# B&R Automation Studio project develop
Automation Studio 4.3.6.57 SP; technology packages: Acp10Arnc0 3.18.2

## Configuration ARM

CPU X20CP0410, AutomationRuntime B4.63, Build 4.1.2, Vc V4.62.0

### Task classes (Cpu.sw)
```
Cyclic#4 (cycle 100000 us, tolerance 100000 us):
  P76C <- P76Sample.P76C.prg
DataObjects: P76config <- Parameter.P76config.dob
Binaries: FWRules, udbdef, TCData, ashwd, ashwac, asfw, iomap, sysconf, Role, User, arconfig
Libraries: Operator, Runtime, AsTime, AsIecCon, brsystem, DataObj, sys_lib, ac_invlib, AsArLog, AsCANopen, AsBrStr, FileIO, AsBrMath, AsEPL
```

### Hardware
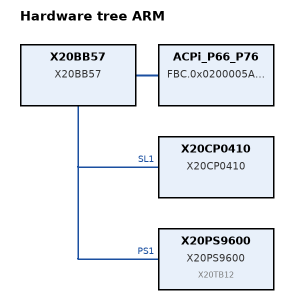
```
ACPi_P66_P76 : FBC.0x0200005A.320.ACPi_P66_P76 v1.3 (OrderNumber=ACPi_P66_P76)  [CAN1 -> X20BB57.IF7]
X20BB57 : X20BB57 v1.1.0.0
  Connector IF7:
    Baudrate = 250000
    ActivateCANIO = 0
    ActivateCanOpen = 1
    p100c_parametervalue = 1000
    p100d_parametervalue = 3
X20CP0410 : X20CP0410 v1.2.0.0  [SL -> X20BB57.SL1]
  Connector IF2:
    ActivateDevice = 1
    Mode = Manual
    InternetAddress = 192.168.0.35
    SubnetMask = 255.255.255.0
  ConfigurationID = develop_ARM
  TimerDeviceType = SWIOTIMER
  Cyclic1Duration = 10000
  Cyclic1Tolerance = 10000
  Cyclic2Duration = 20000
  Cyclic2Tolerance = 20000
  Cyclic3Duration = 50000
  Cyclic3Tolerance = 50000
  Cyclic4Duration = 100000
  Cyclic4Tolerance = 100000
  Cyclic5Duration = 200000
  Cyclic5Tolerance = 200000
  Cyclic6Duration = 500000
  Cyclic6Tolerance = 500000
  Cyclic7Duration = 1000000
  Cyclic7Tolerance = 1000000
  Cyclic8Duration = 10000
  Cyclic8Tolerance = 30000000
X20PS9600 : X20PS9600 v1.2.0.0  [PS -> X20BB57.PS1; SS1 -> X20TB12.SS]
X20TB12 : X20TB12 v1.0.0.0
```

### IoMap.iom - X20CP0410/IoMap.iom
```iecst
VAR_CONFIG
	::P76C:ac_inv_alloc_0.io_mapping.ModuleOK AT %IX."ACPi_P66_P76".ModuleOk;
	::P76C:ac_inv_alloc_0.io_mapping.LCR AT %IW."ACPi_P66_P76".LCR_2002sub5;
	::P76C:ac_inv_alloc_0.io_mapping.OTR AT %IW."ACPi_P66_P76".OTR_2002sub6;
	::P76C:ac_inv_alloc_0.io_mapping.THD AT %IW."ACPi_P66_P76".THD_2002suba;
	::P76C:ac_inv_alloc_0.io_mapping.HMIS AT %IW."ACPi_P66_P76".HMIS_2002sub29;
	::P76C:ac_inv_alloc_0.io_mapping._LFT AT %IW."ACPi_P66_P76".LFT_2029sub16;
	::P76C:ac_inv_alloc_0.io_mapping.THR AT %IW."ACPi_P66_P76".THR_2042sub1f;
	::P76C:ac_inv_alloc_0.io_mapping.CMDD AT %QW."ACPi_P66_P76".CMDD_6040;
	::P76C:ac_inv_alloc_0.io_mapping.ETAD AT %IW."ACPi_P66_P76".ETAD_6041;
	::P76C:ac_inv_alloc_0.io_mapping.LFRD AT %QW."ACPi_P66_P76".LFRD_6042;
	::P76C:ac_inv_alloc_0.io_mapping.RFRD AT %IW."ACPi_P66_P76".RFRD_6044;
END_VAR
```

## Configuration ATOM

CPU X20CP3585, AutomationRuntime L4.10, Build 2.95.3, Vc V4.15.9

### Task classes (Cpu.sw)
```
Cyclic#4:
  P84 <- P84Sample.P84.prg
  P74 <- P74Sample.P74.prg
DataObjects: P84config <- P84Sample.P84config.dob, P74config <- P74Sample.P74config.dob, Acp10sys
Binaries: udbdef, ashwac, ashwd, sysconf, asfw, arconfig, iomap, Acp10cfg, Acp10map, NeueNcMap
Libraries: brsystem, DataObj, sys_lib, ac_invlib, AsEPL, AsArLog, AsBrStr, AsBrMath, Operator, Runtime, AsTime, AsIecCon, asstring, AsCANopen, FileIO, powerlnk, ncglobal, AsUSB, acp10sdc, wh_regl, acp10sim, wh_aclib, acp10par, acp10man
```

### Hardware
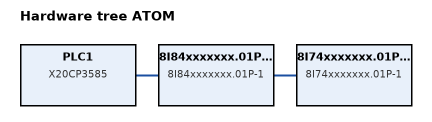
```
8I74xxxxxxx.01P-1 : 8I74xxxxxxx.01P-1 v1.4.0.0  [PLK1 -> 8I84xxxxxxx.01P-1.PLK2 (NodeNumber=10) [Cable Type=PowerlinkCable, Length=10, Version=1.0.0.1]]
  Supervision = off
  packedETAD = packed
  packedETI = packed
  packedCMDD = packed
  packedCMI = packed
  DownloadParameters = no
  ACC = 10
  DEC = 10
8I84xxxxxxx.01P-1 : 8I84xxxxxxx.01P-1 v1.0.9.2  [PLK1 -> PLC1.IF3 (NodeNumber=4) [Cable Type=PowerlinkCable, Length=10, Version=1.0.0.1]; PLK2 -> 8I74xxxxxxx.01P-1.PLK1 (NodeNumber=4) [Cable Type=PowerlinkCable, Length=10, Version=1.0.0.1]]
  Supervision = off
  packedETAD = packed
  packedETI = packed
  packedCMDD = packed
  packedCMI = packed
  DownloadParameters = no
  AUT = 1
PLC1 : X20CP3585 v1.4.2.0
  Connector IF2:
    ActivateDevice = 1
    Mode = Manual
    InternetAddress = 192.168.0.10
    SubnetMask = 255.255.255.0
  Connector IF3:
    InaNodeNumber = 1
  ConfigurationID = develop_ATOM
```

### IoMap.iom - PLC1/IoMap.iom
```iecst
(********************************************************************
 * COPYRIGHT -- Bernecker + Rainer
 ********************************************************************
 * File: IoMap.iom
 * Author: hilchenbachc
 * Created: September 05, 2012
 ********************************************************************
 * IO mapping file
 ********************************************************************)
VAR_CONFIG
	::P84:ac_inv_alloc_0.io_mapping.ModuleOK AT %IX."8I84xxxxxxx.01P-1".ModuleOk;
	P84:ac_inv_alloc_0.io_mapping.ETAD AT %IW."8I84xxxxxxx.01P-1".ETAD_Input;
	P84:ac_inv_alloc_0.io_mapping.HMIS AT %IW."8I84xxxxxxx.01P-1".HMIS_Input;
	P84:ac_inv_alloc_0.io_mapping.LCR AT %IW."8I84xxxxxxx.01P-1".LCR_Input;
	P84:ac_inv_alloc_0.io_mapping.THD AT %IW."8I84xxxxxxx.01P-1".THD_Input;
	P84:ac_inv_alloc_0.io_mapping.THR AT %IW."8I84xxxxxxx.01P-1".THR_Input;
	P84:ac_inv_alloc_0.io_mapping.CMDD AT %QW."8I84xxxxxxx.01P-1".CMDD_Output;
	P84:ac_inv_alloc_0.io_mapping.CMI AT %QW."8I84xxxxxxx.01P-1".CMI_Output;
	P84:ac_inv_alloc_0.io_mapping.LFRD AT %QW."8I84xxxxxxx.01P-1".LFRD_Output;
	P84:ac_inv_alloc_0.io_mapping.LTR AT %QW."8I84xxxxxxx.01P-1".LTR_Output;
	P84:ac_inv_alloc_0.io_mapping.LFT AT %IW."8I84xxxxxxx.01P-1".LFT_Input;
	P84:ac_inv_alloc_0.io_mapping.RFRD AT %IW."8I84xxxxxxx.01P-1".RFRD_Input;
	P84:ac_inv_alloc_0.io_mapping.OTR AT %IW."8I84xxxxxxx.01P-1".OTR_Input;
	P74:ac_inv_alloc_0.io_mapping.ETAD AT %IW."8I74xxxxxxx.01P-1".ETAD_Input;
	P74:ac_inv_alloc_0.io_mapping.HMIS AT %IW."8I74xxxxxxx.01P-1".HMIS_Input;
	P74:ac_inv_alloc_0.io_mapping.LCR AT %IW."8I74xxxxxxx.01P-1".LCR_Input;
	P74:ac_inv_alloc_0.io_mapping.RFRD AT %IW."8I74xxxxxxx.01P-1".RFRD_Input;
	P74:ac_inv_alloc_0.io_mapping.OTR AT %IW."8I74xxxxxxx.01P-1".OTR_Input;
	P74:ac_inv_alloc_0.io_mapping.THD AT %IW."8I74xxxxxxx.01P-1".THD_Input;
	P74:ac_inv_alloc_0.io_mapping.THR AT %IW."8I74xxxxxxx.01P-1".THR_Input;
	P74:ac_inv_alloc_0.io_mapping.LFT AT %IW."8I74xxxxxxx.01P-1".LFT_Input;
	P74:ac_inv_alloc_0.io_mapping.CMDD AT %QW."8I74xxxxxxx.01P-1".CMDD_Output;
	P74:ac_inv_alloc_0.io_mapping.CMI AT %QW."8I74xxxxxxx.01P-1".CMI_Output;
	P74:ac_inv_alloc_0.io_mapping.LFRD AT %QW."8I74xxxxxxx.01P-1".LFRD_Output;
	P74:ac_inv_alloc_0.io_mapping.ModuleOK AT %IX."8I74xxxxxxx.01P-1".ModuleOk;
END_VAR
```

## Logical view

Binary libraries used (declarations not repeated): operator, runtime, AsTime, AsIecCon, brsystem, DataObj, sys_lib, asstring, AsEPL, AsArLog, AsCANopen, AsBrStr, FileIO, AsBrMath

### Package Logical/Libraries - Global libraries

### Library Logical/Libraries/ac_invlib (ANSIC, version 1.10.1) - ACOPOSinverter Library - controls an ACOPOSinverter drive without using the SDC- Library
Depends on: AsEPL, sys_lib, DataObj, AsArLog, brsystem, AsCANopen

#### ac_invlib.typ - Exported data types
```iecst
(********************************************************************
 * COPYRIGHT -- Bernecker + Rainer
 ********************************************************************
 * Library: wh_invlib
 * File: wh_invlib.typ
 * Author: hilchenbachc
 * Created: December 03, 2009
 ********************************************************************
 * Data types of library wh_invlib
 ********************************************************************)

TYPE
	ac_inv_AxIdent : 	STRUCT  (*(internal data type for debugging only !)*)
		p_alloc : REFERENCE TO ac_inv_alloc; (*pointer to fub instance*)
		step_init : UINT; (*initialization step*)
		errorstep : UINT; (*step in which the internal error occured*)
		step_read_data : UINT; (*step for reading data from drive*)
		fub_sdoread : EplSDORead; (*fub instance*)
		fub_sdowrite : EplSDOWrite; (*fub instance*)
		fub_canopen_sdoread : CANopenSDOReadData; (*fub instance*)
		fub_canopen_sdowrite : CANopenSDOWriteData; (*fub instance*)
		node_number : USINT; (*powerlink node number or canopen node number of inverter*)
		interface : STRING[20]; (*interface name*)
		ctrl_on_internal : BOOL; (*internal command for 'ctrl_on'*)
		sdo_read_step : UINT; (*SDORead: step and command interface*)
		sdo_read_par_name : STRING[10]; (*SDORead: name of the inverter parameter*)
		sdo_read_value : UINT; (*SDORead: numeric parameter value*)
		sdo_read_value_constant : STRING[20]; (*SDORead: parameter value constant*)
		sdo_read_status : UINT; (*SDORead: status result*)
		sdo_read_errorinfo : UDINT; (*SDORead: additional error information*)
		sdo_write_step : UINT; (*SDOWrite: step and command interface*)
		sdo_write_par_name : STRING[10]; (*SDOWrite: name of the inverter parameter*)
		sdo_write_value : UINT; (*SDOWrite: numeric parameter value*)
		sdo_write_value_constant : STRING[20]; (*SDOWrite: parameter value constant*)
		sdo_write_status : UINT; (*SDOWrite: status result*)
		sdo_write_errorinfo : UDINT; (*SDOWrite: additional error information*)
		fub_datobjinfo : DatObjInfo; (*fub instance*)
		number_of_parameters : UDINT; (*number of parameters in dataobject*)
		parameterlist_index : UINT; (*parameter list: index of the actual parameter*)
		p_sorted_parameters : ARRAY[0..99]OF UDINT; (*pointer to list with the sorted parameters*)
		dont_sort_parameters : BOOL; (*don't sort parameters from datamodules*)
		write_parameterlist_step : UINT; (*write parameter list: step and command interface*)
		write_parameterlist_status : UINT; (*write parameter list: status result*)
		compare_parameterlist_step : UINT; (* Compare paameterlist: step and command interface *)
		compare_parameterlist_status : UINT; (* Compare parameterlist: status result *)
		compare_parameterlist_index : USINT; (* compare parameterlist: index of the actual parameter *)
		compare_value_constant : STRING[20]; (*SDORead: parameter value constant*)
		log_info : STRING[60]; (*row in logging information*)
		fub_log_write : AsArLogWrite; (*fub instance*)
		kv_old : UINT; (*gain speed controller in %*)
		ti_old : UINT; (*integral time speed controller in %*)
		counter_cyclic_data : USINT; (*cycle counter for cyclic read data*)
		HMIS_old : INT;
		rated_motor_frequency : REAL; (*FrS*)
		rated_motor_speed : REAL; (*nSP*)
		maximum_output_frequency : REAL; (*tFr*)
		polepairs : USINT; (*no of motor polepairs*)
		use_rpm : BOOL; (*1 = use rpm instead Hertz for motor speeds*)
		t_limit_old : ARRAY[0..1]OF REAL;
		cycleTime : REAL; (*cycle time of the task*)
		timer : REAL; (*timer for waiting actions*)
		device_name : STRING[20]; (*Device- Name from Powerlink Object 0x1008*)
		drive_type : USINT; (*0 = unknown, 1 = P84, 2 = P74*)
		isCANopen : BOOL; (*1 = is a CANopen- device*)
		tempUINT : UINT;
	END_STRUCT;
	ac_inv_Mapping : 	STRUCT
		ModuleOK : BOOL; (*Module OK (from drive)*)
		ETAD : UINT; (*Status Word (from drive)*)
		HMIS : UINT; (*Drive state Input (from drive)*)
		RFRD : INT; (*Output- velocity (from drive)*)
		OTR : INT; (*Motor torque (from drive)*)
		LCR : UINT; (*Drive Current (from drive)*)
		THD : UINT; (*Drive Thermal State (from drive)*)
		THR : UINT; (*Motor Thermal State (from drive)*)
		LFT : INT; (*Fault Code ( from drive) as INT for EPL-Mapping*)
		_LFT : UINT; (*Fault Code ( from drive) as UINT for CANopen-Mapping (P84 only)*)
		CMDD : UINT; (*Control Word (to drive)*)
		CMI : UINT; (*Extended Control Word (to drive)*)
		LFRD : INT; (*Speed setpoint (to drive)*)
		LTR : INT; (*Torque setpoint (to drive) (P84 only)*)
	END_STRUCT;
END_TYPE
```

#### ac_invlib.var - Exported constants
```iecst
VAR CONSTANT
	ac_invlibERR_CFI : UINT := 50005; (*one or more parameter were corrected by the drive due to consistency check*)
	ac_invlibERR_WRONG_ARVERSION : UINT := 50003; (*wrong Automation Runtime version*)
	ac_invlibERR_PARNOTFOUND : UINT := 50002; (*wrong parameter name*)
	ac_invlibERR_ILLEGAL_AXIDENT : UINT := 50001; (*invalid ax_ident*)
	ac_invlibERR_NETWORK : UINT := 50004; (*network timeout*)
END_VAR
```

#### ac_invlib.fun - Exported functions and function blocks
```iecst
FUNCTION_BLOCK ac_inv_alloc (*axis allocation*)
	VAR_INPUT
		pDevice : UDINT; (*pointer to name of device i.e. 'IF3.ST4'*) (* *) (*#PAR*)
		pcfgpar : ARRAY[0..2] OF UDINT; (*pointer to name of parameter data objects*) (* *) (*#PAR*)
		io_mapping : ac_inv_Mapping; (*IO- mapping (must be connected in physical view)*) (* *) (*#PAR*)
		rpm : BOOL; (*use rpm instead of Hertz for n_set and n_act*) (* *) (*#PAR#OPT*)
		no_parameter_sort : BOOL; (*1 = don't sort parameters from datamodules*) (* *) (*#PAR#OPT*)
	END_VAR
	VAR_OUTPUT
		status : UINT; (*fub status*) (* *) (*#CYC*)
		message : STRING[80]; (*error message, when allocation fails*) (* *) (*#CYC*)
		ax_ident : UDINT; (*axis identifier ('handle') for function blocks*) (* *) (*#CYC*)
	END_VAR
END_FUNCTION_BLOCK

FUNCTION_BLOCK ac_inv (*cyclic execution*)
	VAR_INPUT
		ax_ident : UDINT; (*axis identifier (handle) from ac_inv_alloc()*) (* *) (*#PAR*)
		quickstop : BOOL; (*0 = perform fast stop*) (* *) (*#CMD*)
		ctrl_on : BOOL; (*switch controller (power stage) on/off*) (* *) (*#CMD*)
		f_quit : BOOL; (*quit inverter fault*) (* *) (*#CMD*)
		kv : UINT; (*gain speed controller in %*) (* *) (*#OPT#CYC*)
		ti : UINT; (*Integral time speed controller in %*) (* *) (*#OPT#CYC*)
		n_set : REAL; (*set speed (% of tFr or rpm)*) (* *) (*#CYC*)
		t_set : REAL; (*set torque in % nominal motor torque (P84 only)*) (* *) (*#OPT#CYC*)
		t_limit : ARRAY[0..1] OF REAL; (*torque limit*) (* *) (*#OPT#CYC*)
		write_parameter : USINT; (*write a parameter to the drive (see 'parameter_name' and 'parameter_value')*) (* *) (*#CMD#OPT*)
		read_parameter : USINT; (*read a parameter from the drive (see 'parameter_name' and 'parameter_value')*) (* *) (*#CMD#OPT*)
		parameter_name : STRING[4]; (*name of the inverter parameter to be written or to be read*) (* *) (*#PAR#OPT*)
		parameter_value : STRING[15]; (*value of the inverter parameter to be written or to be read*) (* *) (*#CMD#OPT*)
		C211 : BOOL; (*Control Bit*) (* *) (*#OPT#CYC*)
		C212 : BOOL; (*Control Bit*) (* *) (*#OPT#CYC*)
		C213 : BOOL; (*Control Bit*) (* *) (*#OPT#CYC*)
		C214 : BOOL; (*Control Bit*) (* *) (*#OPT#CYC*)
		C215 : BOOL; (*Control Bit*) (* *) (*#OPT#CYC*)
		activate_tuning : BOOL; (*1 = set motor tuning active. tuning will be activated with 'ctrl_on=true'*) (* *) (*#OPT#CYC*)
	END_VAR
	VAR_OUTPUT
		ctrl_ready : BOOL; (*controller is ready to be switched on*) (* *) (*#CYC*)
		power_line : BOOL; (*power line present = 1*) (* *) (*#CYC*)
		ctrl_is_on : BOOL; (*controller (power stage) is on/off*) (* *) (*#CYC*)
		initialized : BOOL; (*drive initialized*) (* *) (*#CYC*)
		alarm : BOOL; (*alarm*) (* *) (*#CYC*)
		fault : BOOL; (*inverter fault see 'fault code'*) (* *) (*#CYC*)
		PRA_detected : BOOL; (*Power removal (PRA) was detected -> reset ctrl_on*) (* *) (*#CYC#OPT*)
		n_act : REAL; (*actual speed (% of tFr or rpm)*) (* *) (*#CYC*)
		t_act : REAL; (*torque in % of nominal motor torque*) (* *) (*#CYC*)
		current : REAL; (*current in A*) (* *) (*#CYC*)
		thst_drive : REAL; (*thermal state drive in %*) (* *) (*#CYC#OPT*)
		thst_motor : REAL; (*thermal state motor in %*) (* *) (*#CYC*)
		udc : REAL; (*dc voltage in V*) (* *) (*#CYC*)
		encoder_value : UINT; (*encoder value (P84 only)*) (* *) (*#CYC#OPT*)
		drive_state : STRING[4]; (*drive state*) (* *) (*#CYC*)
		fault_code : STRING[4]; (*fault code (LFT) as string*) (* *) (*#CYC*)
		LFT : UINT; (*LFT*) (* *) (*#CYC*)
		status : UINT; (*fub status*) (* *) (*#CYC*)
	END_VAR
END_FUNCTION_BLOCK
```

#### ac_inv_global.h
```c
#ifndef _AC_INV_GLOBAL_H
#define _AC_INV_GLOBAL_H

#include <bur/plctypes.h>
#include <ac_invlib.h>
#include <ctype.h>
#include <string.h>
#include <math.h>

#define STEP_W_NETWORK					0
#define STEP_READ_DEVICE_NAME			1
#define STEP_LOG_DEVICE_TYPE			200
#define STEP_W_LOG_DEVICE_TYPE			201
#define STEP_W_FACTORY_RESET_P74		202
#define STEP_W_P74_CONFIG_1				203
#define STEP_W_P74_CONFIG_2				204
#define STEP_W_FACTORY_RESET_P84		3
#define STEP_W_P84_CONFIG_1				4
#define STEP_W_P84_CONFIG_2				5
#define STEP_W_REFERENCE_CHANNEL_SET 	9
#define STEP_W_PARAMETER_LIST_DOWNLOAD	10
#define STEP_CHECK_PARAMETER_LIST		20
#define STEP_W_PARAMETER_LIST_CHECKED	22
#define STEP_READ_KV					30
#define STEP_READ_TI					31
#define STEP_READ_OUTPUT_FREQUENCY		32
#define STEP_READ_TORQUE_LIMIT_0		33
#define STEP_READ_TORQUE_LIMIT_1		34
#define STEP_READ_CTT					40
#define STEP_READ_RATED_FREQ			41
#define STEP_READ_RATED_SPEED			42
#define STEP_W_READ_RATED_SPEED			43
#define STEP_W_COMMAND					100
#define STEP_P84_WRITE_TUN				300
#define STEP_W_P84_TUNING_DONE			310
#define STEP_P74_START_TUNING			350
#define STEP_P74_TUNING_1				360
#define STEP_P74_TUNING_2				361
#define STEP_P74_TUNING_3				362
#define STEP_P74_TUNING_4				363
#define STEP_P74_TUNING_5				364
#define STEP_P74_TUNING_6				365
#define STEP_P74_TUNING_7				366
#define STEP_P74_TUNING_8				367

#define STEP_INTERNAL_ERROR				9999

char * m_ltoa(long value, char *string, int radix);
long m_atol(char*);
/*int strcasecmp( char *s1, char *s2 );*/
int find_parameter( char *name, UINT *index, USINT *subindex, USINT drive_type );
int find_download_index( char *name,  USINT drive_type );
char *find_value_constant( char *name, UINT value, USINT drive_type );
int find_numeric_value( char *name, char *constant, USINT drive_type );
void read_parameter( ac_inv_AxIdent *ax_ident );
void write_parameter( ac_inv_AxIdent *ax_ident );
void write_parameterlist( ac_inv_AxIdent *ax_ident );
void compare_parameterlist( ac_inv_AxIdent *ax_ident );
void logCOF( ac_inv_AxIdent *ax_ident );
void sort_parameterlist( ac_inv_AxIdent *ax_ident );
void create_parameterlist( ac_inv_AxIdent *ax_ident );
#endif
```

#### ac_invhelp.c
```c
#include <bur/plctypes.h>
#include <ctype.h>

/* long to ascii conversion */
char * m_ltoa(long value, char *string, int radix)
{
  char tmp[33];
  char *tp = tmp;
  long i;
  unsigned long v;
  int sign;

  if (radix > 36 || radix <= 1)
  {
    return 0;
  }

  sign = (radix == 10 && value < 0);
  if (sign)
    v = -value;
  else
    v = (unsigned long)value;
  while (v || tp == tmp)
  {
    i = v % radix;
    v = v / radix;
    if (i < 10)
      *tp++ = i+'0';
    else
      *tp++ = i + 'a' - 10;
  }

  if (sign)
    *string++ = '-';
  while (tp > tmp)
    *string++ = *--tp;
  *string = 0;
  return string;
}

long m_atol( char* s ){
	long l = 0;
	int sign = 0;

	while( *s ){
		if( *s  == '-' ){
			if( sign == 0 )
				sign = -1;
			else
				return 0; /* error: more than one sign */
		}
		if( *s == '+' ){
			if( sign == 0 )
				sign = +1;
			else
				return 0; /* error: more than one sign */
		}
		if( *s >= '0' && *s <= '9' ){
			l *= 10;
			l += *s - '0';
		}
		++s;
	}
	if( sign < 0 )
		l = -l;
	return l;
}

/* case insensitive string comparator */
int strcasecmp( char *s1, char *s2 ){
	do{
		if( tolower( *s1 ) != tolower( *s2 ) ){
			return ( *s1 - *s2 );
		}
		++s1;
		++s2;
	} while (*s1 && *s2);
	if( *s1 != *s2 ) /* different length */
		return -1;

	return 0;
}
```

#### ac_invparameter.c
```c
#include <bur/plctypes.h>
#include <stdlib.h>
#include <string.h>
#include <ac_inv_global.h>

#include <ac_invparameter.h>
#include <P84_registers.h>
#include <P74_registers.h>

/* -----------------------------------------------------------------------------------
   find parameter in list
   returns index of parameter in parameter list or -1 in case of failure
   -----------------------------------------------------------------------------------
*/

int find_parameter( char *name, UINT *index, USINT *subindex, USINT drive_type )
{
	int i = 0;
	acpireg *regs = drive_type == 2 ? p74reg : p84reg;

	while( regs[i].name )
	{
		if( strcasecmp( regs[i].name, name ) == 0 )   /* found ? */
		{
			if( index )
				*index = regs[i].index;
			if( subindex )
				*subindex = regs[i].subindex;
			return i;
		}
		++i;
	}
	return -1; /* not found */
}

/* -----------------------------------------------------------------------------------
 	returns the download index of a parameter or -1 in case of failure
   -----------------------------------------------------------------------------------
*/

int find_download_index( char *name,  USINT drive_type )
{
	int i = 0;
	char **list = drive_type == 2 ? P74_download_index : P84_download_index;

	while( list[i] )
	{
		if( strcasecmp(  list[i], name ) == 0 )   /* found ? */
		{
			return i;
		}
		++i;
	}
	return -1; /* not found */
}

/* -----------------------------------------------------------------------------------
 	returns the enumerated name of the parameter's value
   -----------------------------------------------------------------------------------
*/

char *find_value_constant( char *name, UINT value, USINT drive_type )
{
	int index;
	static char s[20];
	char sign = 'u';
	acpireg *regs = drive_type == 2 ? p74reg : p84reg;

	index = find_parameter( name, 0, 0, drive_type );
	if( index >= 0 )
	{
		int i = 0;
		sign = regs[index].sign;
		/* translate parameter value to enumeration constant */
		if( regs[index].enu )   /* are constants defined ? */
		{
			while( regs[index].enu[i].name )
			{
				if( regs[index].enu[i].value == value )
				{
					return( regs[index].enu[i].name );  /* return enumerated name */
				}
				++i;
			}
		}
	}
	if( sign == 'u' )
		m_ltoa( value , s, 10 );  /* return numeric value */
	else
		m_ltoa( (INT) value, s, 10 );
	return s; /* not found or no constant defined */

}

/* -----------------------------------------------------------------------------------
 	returns the value for the given constant
   -----------------------------------------------------------------------------------
*/

int find_numeric_value( char *name, char *constant, USINT drive_type )
{
	int index;
	acpireg *regs = drive_type == 2 ? p74reg : p84reg;

	index = find_parameter( name, 0, 0, drive_type );
	if( index >= 0 )
	{
		int i = 0;
		/* try to find the constant */
		if( regs[index].enu )   /* are constants defined ? */
		{
			while( regs[index].enu[i].name )
			{
				if( strcasecmp( regs[index].enu[i].name, constant ) == 0 )
				{
					return( regs[index].enu[i].value );  /* return enumerated name */
				}
				++i;
			}
		}
	}
	return m_atol(constant);  /* return numeric value */

}

/* -------------------------------------------------------------------------------------
   read parameter from inverter
   -------------------------------------------------------------------------------------
*/

void read_parameter( ac_inv_AxIdent *ax_ident )
{

	for(;;)
	{
		switch( ax_ident->sdo_read_step )
		{
		case 0: /* wait for command */
			ax_ident->fub_sdoread.enable = 0;
			break;

		case 1: /* start read */
			if( find_parameter( ax_ident->sdo_read_par_name, &ax_ident->fub_sdoread.index, &ax_ident->fub_sdoread.subindex, ax_ident->drive_type ) < 0 )
			{
				ax_ident->sdo_read_step = 3;
				ax_ident->sdo_read_status = ac_invlibERR_PARNOTFOUND;
				ax_ident->sdo_read_errorinfo = 0;
				continue; /* save on cycle */
			}
			else
			{
				/* fill the fub structure */
				ax_ident->sdo_read_value = 0;
				ax_ident->fub_sdoread.enable = 1;
				ax_ident->fub_sdoread.pData = (UDINT) &ax_ident->sdo_read_value;
				ax_ident->fub_sdoread.datalen = sizeof(ax_ident->sdo_read_value);
				ax_ident->sdo_read_step = 2;
				ax_ident->sdo_read_status = 65535;
				ax_ident->sdo_read_errorinfo = 0;

			}
			break;

		case 2: /* wait until read */
			if( ax_ident->fub_sdoread.status != 65535 )  /* value read */
			{
				ax_ident->fub_sdoread.enable = 0; /* disable fub */
				ax_ident->sdo_read_status = ax_ident->fub_sdoread.status;
				ax_ident->sdo_read_errorinfo = ax_ident->fub_sdoread.errorinfo;
				ax_ident->sdo_read_step = 3;
				continue; /* save on cycle */
			}
			break;

		case 3: /* write into log */
		{
			char tempstring[20];
			const char *ret = find_value_constant( ax_ident->sdo_read_par_name, ax_ident->sdo_read_value, ax_ident->drive_type );
			strcpy( ax_ident->sdo_read_value_constant, ret );
			strcpy( ax_ident->log_info, ax_ident->interface );
			strcat( ax_ident->log_info, "." );
			m_ltoa( ax_ident->node_number, tempstring, 10 );
			strcat( ax_ident->log_info, tempstring );
			strcat( ax_ident->log_info, "  " );
			strcat( ax_ident->log_info, ax_ident->sdo_read_par_name );
			strcat( ax_ident->log_info, " -->#" );
			strcat( ax_ident->log_info, ax_ident->sdo_read_value_constant );
			if( ax_ident->sdo_read_status != 0 )
			{
				ax_ident->fub_log_write.logLevel = arlogLEVEL_FATAL;
				if( ax_ident->sdo_read_status == ERR_ASEPL_ACCESS_FAILED )
				{
					strcat( ax_ident->log_info, ":errorinfo=" );
					strcat( ax_ident->log_info, "/0x" );
					m_ltoa( ax_ident->sdo_read_errorinfo, tempstring, 16 );
					strcat( ax_ident->log_info, tempstring );
				}
				else if( ax_ident->sdo_read_status == ac_invlibERR_PARNOTFOUND )
				{
					strcat( ax_ident->log_info, ":parameter not found" );
				}
			}
			else
			{
				ax_ident->fub_log_write.logLevel = arlogLEVEL_INFO;
			}
			ax_ident->fub_log_write.errornr = ax_ident->sdo_read_status;
			ax_ident->fub_log_write.mem = (UDINT) &ax_ident->node_number;
			ax_ident->fub_log_write.len = sizeof(ax_ident->node_number);
			ax_ident->fub_log_write.asciiString = (UDINT) ax_ident->log_info;
			AsArLogWrite( &ax_ident->fub_log_write );
			ax_ident->sdo_read_step = 4;
		}
		break;

		case 4:  /* wait until log entry written */
			if( ax_ident->fub_log_write.status != 65535 )
			{
				ax_ident->sdo_read_step = 0;
			}
			else
			{
				AsArLogWrite( &ax_ident->fub_log_write );
			}
			break;

			/* start reading without writing to log file in case of success (for fub inside use ! */
		case 10:
			if( find_parameter( ax_ident->sdo_read_par_name, &ax_ident->fub_sdoread.index, &ax_ident->fub_sdoread.subindex, ax_ident->drive_type ) < 0 )
			{
				ax_ident->sdo_read_step = 3;
				ax_ident->sdo_read_status = ac_invlibERR_PARNOTFOUND;
				ax_ident->sdo_read_errorinfo = 0;
				continue; /* save on cycle */
			}
			else
			{
				/* fill the fub structure */
				ax_ident->sdo_read_value = 0;
				ax_ident->fub_sdoread.enable = 1;
				ax_ident->fub_sdoread.pData = (UDINT) &ax_ident->sdo_read_value;
				ax_ident->fub_sdoread.datalen = sizeof(ax_ident->sdo_read_value);
				ax_ident->sdo_read_step = 11;
				ax_ident->sdo_read_status = 65535;
				ax_ident->sdo_read_errorinfo = 0;
			}
			break;

		case 11: /* wait until read */
			if( ax_ident->fub_sdoread.status != 65535 )  /* value read */
			{
				ax_ident->fub_sdoread.enable = 0; /* disable fub */
				ax_ident->sdo_read_status = ax_ident->fub_sdoread.status;
				ax_ident->sdo_read_errorinfo = ax_ident->fub_sdoread.errorinfo;
				ax_ident->sdo_read_step = 0;
			}
			break;

			/* use SDO read directly (for fub inside use !) */
		case 100:
			ax_ident->fub_sdoread.enable = 1;
			ax_ident->sdo_read_step = 101;
			break;

		case 101:
			if( ax_ident->fub_sdoread.status != 65535 )  /* value read */
			{
				ax_ident->fub_sdoread.enable = 0; /* disable fub */
				ax_ident->sdo_read_status = ax_ident->fub_sdoread.status;
				ax_ident->sdo_read_errorinfo = ax_ident->fub_sdoread.errorinfo;
				ax_ident->sdo_read_step = 0;
			}
			break;

		}
		break;  /* exit for(;;) */
	}

	if( ax_ident->isCANopen )
	{
		/* FUB- Eingaenge umkopieren */
		ax_ident->fub_canopen_sdoread.enable = ax_ident->fub_sdoread.enable;
		ax_ident->fub_canopen_sdoread.index = ax_ident->fub_sdoread.index;
		ax_ident->fub_canopen_sdoread.subindex = ax_ident->fub_sdoread.subindex;
		CANopenSDOReadData( &ax_ident->fub_canopen_sdoread );
		/* FUB- Ausgaenge umkopieren */
		ax_ident->fub_sdoread.status = ax_ident->fub_canopen_sdoread.status;
		ax_ident->fub_sdoread.errorinfo = ax_ident->fub_canopen_sdoread.errorinfo;
	}
	else
		EplSDORead( &ax_ident->fub_sdoread );

}

/* -------------------------------------------------------------------------------------
   write parameter to inverter via EPL
   -------------------------------------------------------------------------------------
*/

void write_parameter( ac_inv_AxIdent *ax_ident )
{

	for(;;)
	{
		switch( ax_ident->sdo_write_step )
		{
		case 0: /* wait for command */
			ax_ident->fub_sdowrite.enable = 0;
			break;

		case 1: /* start write */
			if( find_parameter( ax_ident->sdo_write_par_name, &ax_ident->fub_sdowrite.index, &ax_ident->fub_sdowrite.subindex, ax_ident->drive_type ) < 0 )
			{
				ax_ident->sdo_write_step = 3;
				ax_ident->sdo_write_status = ac_invlibERR_PARNOTFOUND;
				ax_ident->sdo_write_errorinfo = 0;
				continue; /* save on cycle */
			}
			else
			{
				/* fill the fub structure */
				ax_ident->sdo_write_value = find_numeric_value( ax_ident->sdo_write_par_name, ax_ident->sdo_write_value_constant, ax_ident->drive_type );
				ax_ident->fub_sdowrite.enable = 1;
				ax_ident->sdo_write_step = 2;
				ax_ident->sdo_write_status = 65535;
				ax_ident->sdo_write_errorinfo = 0;
			}
			break;

		case 2: /* wait until written */
			if( ax_ident->fub_sdowrite.status != 65535 )
			{
				ax_ident->sdo_write_status = ax_ident->fub_sdowrite.status;
				ax_ident->sdo_write_errorinfo = ax_ident->fub_sdowrite.errorinfo;
				ax_ident->fub_sdowrite.enable = 0; /* disable fub */
				ax_ident->sdo_write_step = 3;
				continue; /* save on cycle */
			}
			break;

		case 3: /* write into log */
		{
			char tempstring[20];

			strcpy( ax_ident->log_info, ax_ident->interface );
			strcat( ax_ident->log_info, "." );
			m_ltoa( ax_ident->node_number, tempstring, 10 );
			strcat( ax_ident->log_info, tempstring );
			strcat( ax_ident->log_info, " #" );
			strcat( ax_ident->log_info, ax_ident->sdo_write_value_constant );
			strcat( ax_ident->log_info, " -->" );
			strcat( ax_ident->log_info, ax_ident->sdo_write_par_name );
			if( ax_ident->sdo_write_status != 0 )
			{
				if( ax_ident->sdo_write_status == ERR_ASEPL_ACCESS_FAILED )
				{
					ax_ident->fub_log_write.logLevel = arlogLEVEL_FATAL;
					strcat( ax_ident->log_info, " :errorinfo=" );
					strcat( ax_ident->log_info, "/0x" );
					m_ltoa( ax_ident->sdo_write_errorinfo, tempstring, 16 );
					strcat( ax_ident->log_info, tempstring );
				}
				else if( ax_ident->sdo_write_status == ac_invlibERR_PARNOTFOUND )
				{
					strcat( ax_ident->log_info, ":parameter not found" );
				}
			}
			else
			{
				ax_ident->fub_log_write.logLevel = arlogLEVEL_INFO;
			}
			ax_ident->fub_log_write.errornr = ax_ident->sdo_write_status;
			ax_ident->fub_log_write.mem = (UDINT) &ax_ident->node_number;
			ax_ident->fub_log_write.len = sizeof(ax_ident->node_number);
			ax_ident->fub_log_write.asciiString = (UDINT) ax_ident->log_info;
			AsArLogWrite( &ax_ident->fub_log_write );
			ax_ident->sdo_write_step = 4;
			continue; /* save on cycle */
		}
		break;

		case 4:  /* wait until log entry written */
			if( ax_ident->fub_log_write.status != 65535 )
			{
				ax_ident->sdo_write_step = 0;
			}
			else
			{
				AsArLogWrite( &ax_ident->fub_log_write );
			}
			break;

		}
		break; /* exit for(;;) */
	}

	if( ax_ident->isCANopen )
	{
		/* FUB- Eingaenge umkopieren */
		ax_ident->fub_canopen_sdowrite.enable = ax_ident->fub_sdowrite.enable;
		ax_ident->fub_canopen_sdowrite.index = ax_ident->fub_sdowrite.index;
		ax_ident->fub_canopen_sdowrite.subindex = ax_ident->fub_sdowrite.subindex;
		CANopenSDOWriteData( &ax_ident->fub_canopen_sdowrite );
		/* FUB- Ausgaenge umkopieren */
		ax_ident->fub_sdowrite.status = ax_ident->fub_canopen_sdowrite.status;
		ax_ident->fub_sdowrite.errorinfo = ax_ident->fub_canopen_sdowrite.errorinfo;
	}
	else
		EplSDOWrite( &ax_ident->fub_sdowrite );

}

/* -------------------------------------------------------------------------------------
   write parameter from parameter list to inverter
   -------------------------------------------------------------------------------------
*/

void write_parameterlist( ac_inv_AxIdent *ax_ident )
{
	char tempstring[80];
	char *source, *dest;
	int i;

	switch( ax_ident->write_parameterlist_step )
	{
	case 0:
		break;

	case 1: /* download started - write header to log */
		if( ax_ident->p_alloc->pcfgpar[0] || ax_ident->p_alloc->pcfgpar[1] || ax_ident->p_alloc->pcfgpar[2] )
		{
			ax_ident->parameterlist_index = 0;
			ax_ident->sdo_write_status = 0; /* clear last SDO write error */
			strcpy( ax_ident->log_info, ax_ident->interface );
			strcat( ax_ident->log_info, "." );
			m_ltoa( ax_ident->node_number, tempstring, 10 );
			strcat( ax_ident->log_info, tempstring );
			strcat( ax_ident->log_info, " download " );
			for( i = 0; i < 3; ++i )
			{
				if( ax_ident->p_alloc->pcfgpar[i] )
				{
					strcat( ax_ident->log_info, " \"" );
					strcat( ax_ident->log_info, (char*)	ax_ident->p_alloc->pcfgpar[i] );
					strcat( ax_ident->log_info, "\" " );
				}
			}
			ax_ident->fub_log_write.logLevel = arlogLEVEL_INFO;
			ax_ident->fub_log_write.errornr = 0;
			ax_ident->fub_log_write.mem = (UDINT) &ax_ident->node_number;
			ax_ident->fub_log_write.len = sizeof(ax_ident->node_number);
			ax_ident->fub_log_write.asciiString = (UDINT) ax_ident->log_info;
			AsArLogWrite( &ax_ident->fub_log_write );
			ax_ident->write_parameterlist_step	= 2;
		}
		else
		{
			ax_ident->write_parameterlist_step	= 0;
		}
		break;

	case 2:  /* wait until log entry written */
		if( ax_ident->fub_log_write.status == 0 )
		{
			ax_ident->write_parameterlist_step = 3;
		}
		else if( ax_ident->fub_log_write.status != 65535 )  /* error */
		{
			ax_ident->write_parameterlist_step = 0;
		}
		else
		{
			AsArLogWrite( &ax_ident->fub_log_write );
		}
		break;

	case 3: /* read next row */
		if( ax_ident->sdo_write_step == 0 )   /* service channel free ? */
		{
			source = (char*) ax_ident->p_sorted_parameters[ax_ident->parameterlist_index];
			dest = tempstring;
			memset( tempstring, 0, sizeof(tempstring) );
			if( ax_ident->sdo_write_status != 0 )  /* error after writing the last parameter */
			{
				ax_ident->write_parameterlist_status = ax_ident->sdo_write_status;
				ax_ident->write_parameterlist_step = 0;
				break;
			}
			else if( ax_ident->parameterlist_index >= ax_ident->number_of_parameters )  /* end of list */
			{
				strcpy( ax_ident->log_info, ax_ident->interface );
				strcat( ax_ident->log_info, "." );
				m_ltoa( ax_ident->node_number, tempstring, 10 );
				strcat( ax_ident->log_info, tempstring );
				strcat( ax_ident->log_info, " end of " );
				for( i = 0; i < 3; ++i )
				{
					if( ax_ident->p_alloc->pcfgpar[i] )
					{
						strcat( ax_ident->log_info, " \"" );
						strcat( ax_ident->log_info, (char*)	ax_ident->p_alloc->pcfgpar[i] );
						strcat( ax_ident->log_info, "\" " );
					}
				}
				ax_ident->fub_log_write.logLevel = arlogLEVEL_INFO;
				ax_ident->fub_log_write.errornr = 0;
				ax_ident->fub_log_write.mem = (UDINT) &ax_ident->node_number;
				ax_ident->fub_log_write.len = sizeof(ax_ident->node_number);
				ax_ident->fub_log_write.asciiString = (UDINT) ax_ident->log_info;
				AsArLogWrite( &ax_ident->fub_log_write );
				ax_ident->write_parameterlist_step	= 4;
				break;
			}
			else
			{
				while( ax_ident->parameterlist_index < ax_ident->number_of_parameters )
				{
					if( *source == 0 )   /* end of a row ? */
					{
						strncpy( ax_ident->sdo_write_value_constant, tempstring, sizeof(ax_ident->sdo_write_value_constant) - 1 );
						ax_ident->sdo_write_step = 1;  /* write parameter to inverter */
						++ax_ident->parameterlist_index;
						break;
					}
					else if( !isprint(*source) || *source == ' ' )   /* ignore control chars and spaces */
					{
						++source;
					}
					else if( *source == '=' )
					{
						++source;
						strncpy( ax_ident->sdo_write_par_name, tempstring, sizeof(ax_ident->sdo_write_par_name) - 1 );
						memset( tempstring, 0, sizeof(tempstring) );
						dest = tempstring;
					}
					else
					{
						*dest++ = *source++; /* copy to tempstring */
					}
				}
			}
		}
		break;

	case 4: /* wait until tail is written */
		if( ax_ident->fub_log_write.status != 65535 )
		{
			ax_ident->write_parameterlist_step = 0;
		}
		else
		{
			AsArLogWrite( &ax_ident->fub_log_write );
		}
		break;

	}

}

/* -------------------------------------------------------------------------------------
   compare parameter from parameter list with inverter
   -------------------------------------------------------------------------------------
*/

void compare_parameterlist( ac_inv_AxIdent *ax_ident )
{
	char tempstring[80];
	char *source, *dest;

	switch( ax_ident->compare_parameterlist_step )
	{
	case 0:

		break;

	case 1: /* start comparing */
		ax_ident->parameterlist_index = 0;
		ax_ident->compare_parameterlist_step = 2;
		break;

		/* compare next parameter */
	case 2:
		if( ax_ident->parameterlist_index >= ax_ident->number_of_parameters )  /* end of list */
		{
			ax_ident->compare_parameterlist_step	= 0;
			break;
		}
		else
		{
			source = (char*) ax_ident->p_sorted_parameters[ax_ident->parameterlist_index];
			dest = tempstring;
			memset( tempstring, 0, sizeof(tempstring) );
			while( ax_ident->parameterlist_index < ax_ident->number_of_parameters )
			{
				if( *source == 0 )   /* end of a row ? */
				{
					*dest++ = *source++;
					strncpy( ax_ident->compare_value_constant, tempstring, sizeof(ax_ident->compare_value_constant) - 1 );
					ax_ident->sdo_read_step = 10; /* read without logger entry */
					++ax_ident->parameterlist_index;
					ax_ident->compare_parameterlist_step = 3;
					break;
				}
				else if( !isprint(*source) || *source == ' ' )   /* ignore control chars and spaces */
				{
					++source;
				}
				else if( *source == '=' )
				{
					++source;
					strncpy( ax_ident->sdo_read_par_name, tempstring, sizeof(ax_ident->sdo_read_par_name) - 1 );
					memset( tempstring, 0, sizeof(tempstring) );
					dest = tempstring;
				}
				else
				{
					*dest++ = *source++; /* copy to tempstring */
				}

			}
		}
		break;

		case 3: /* wait for sdo read value */
			if( ax_ident->sdo_read_step == 0 )   /* service channel free ? */
			{
				const char *ret = find_value_constant( ax_ident->sdo_read_par_name, ax_ident->sdo_read_value, ax_ident->drive_type );
				strcpy( ax_ident->sdo_read_value_constant, ret );
				if( strcasecmp( ax_ident->sdo_read_value_constant, ax_ident->compare_value_constant) )  /* different to set value ? */
				{
					ax_ident->compare_parameterlist_step = 4;
				}
				else   /* equal -> ok */
				{
					ax_ident->compare_parameterlist_step = 2;
				}
			}
			break;

		case 4:  /* write into log */
		{
			char tempstring[20];

			strcpy( ax_ident->log_info, ax_ident->interface );
			strcat( ax_ident->log_info, "." );
			m_ltoa( ax_ident->node_number, tempstring, 10 );
			strcat( ax_ident->log_info, tempstring );
			strcat( ax_ident->log_info, "  " );
			strcat( ax_ident->log_info, ax_ident->sdo_read_par_name );
			strcat( ax_ident->log_info, " -->#" );
			strcat( ax_ident->log_info, ax_ident->sdo_read_value_constant );
			strcat( ax_ident->log_info, " (#" );
			strcat( ax_ident->log_info, ax_ident->compare_value_constant );
			strcat( ax_ident->log_info, ")" );
			ax_ident->fub_log_write.logLevel = arlogLEVEL_WARNING;
			ax_ident->fub_log_write.errornr = ac_invlibERR_CFI;
			ax_ident->fub_log_write.mem = (UDINT) &ax_ident->node_number;
			ax_ident->fub_log_write.len = sizeof(ax_ident->node_number);
			ax_ident->fub_log_write.asciiString = (UDINT) ax_ident->log_info;
			AsArLogWrite( &ax_ident->fub_log_write );
			ax_ident->compare_parameterlist_step = 5;
			break;

			case 5:  /* wait until log entry written */
				if( ax_ident->fub_log_write.status != 65535 )
				{
					ax_ident->compare_parameterlist_step = 0;
				}
				else
				{
					AsArLogWrite( &ax_ident->fub_log_write );
				}
			}
			break;

		}

	}

/* -------------------------------------------------------------------------------------
   create a list of parameters from the data modules
   -------------------------------------------------------------------------------------
*/

void create_parameterlist( ac_inv_AxIdent *ax_ident )
{
	int index_module = 0;
	ax_ident->number_of_parameters = 0;
	memset( &ax_ident->p_sorted_parameters, 0, sizeof(ax_ident->p_sorted_parameters) );
	while( ax_ident->p_alloc->pcfgpar[index_module] )
	{
		ax_ident->fub_datobjinfo.enable = 1;
		ax_ident->fub_datobjinfo.pName = ax_ident->p_alloc->pcfgpar[index_module];
		DatObjInfo( &ax_ident->fub_datobjinfo );
		if( ax_ident->fub_datobjinfo.status == 0 )
		{
			char *source = (char*) ax_ident->fub_datobjinfo.pDatObjMem;
			while( ax_ident->fub_datobjinfo.len ){
				if( *source == 0 ){  /* end of a row ? */
					++ax_ident->number_of_parameters;
					while( *source == 0 && ax_ident->fub_datobjinfo.len ){  /* ignore filling zeros */
						++source;
						--ax_ident->fub_datobjinfo.len;
					}
				}
				else if( ax_ident->p_sorted_parameters[ax_ident->number_of_parameters] == 0 ) {  /* store pointer to parameter row */
					ax_ident->p_sorted_parameters[ax_ident->number_of_parameters] = (UDINT) source++;
					ax_ident->fub_datobjinfo.len--;
				}
				else {
					source++;
					ax_ident->fub_datobjinfo.len--;
				}
			}
		}
		if( ++index_module >= 3	)  /* no more data modules */
			break;
	}
}

/* -------------------------------------------------------------------------------------
   compare function for qsort()
   -------------------------------------------------------------------------------------
*/

int compare_download_index_P84 (const void * a, const void * b)
{
	char name[20];
	char *s, *d;
	int index_a=0, index_b=0;
	char **list;

	/* copy parameter name a */
	s = *(char**) a; d= name;
	while( *s != ' ' && *s != 0 && *s != '=')
		*d++ = *s++;
	*d = 0;

	list = P84_download_index;
	while( list[index_a] )
	{
		if( strcasecmp(  list[index_a], name ) == 0 )   /* found ? */
			break;
		++index_a;
	}

	/* copy parameter name b */
	s = *(char**) b; d= name;
	while( *s != ' ' && *s != 0 && *s != '=')
		*d++ = *s++;
	*d = 0;

	list = P84_download_index;
	while( list[index_b] )
	{
		if( strcasecmp(  list[index_b], name ) == 0 )   /* found ? */
			break;
		++index_b;
	}

	if ( index_a <  index_b ) return -1;
	if ( index_a >  index_b ) return 1;

	return 0;
}

int compare_download_index_P74 (const void * a, const void * b)
{
	char name[20];
	char *s, *d;
	int index_a=0, index_b=0;
	char **list;

	/* copy parameter name a */
	s = *(char**) a; d= name;
	while( *s != ' ' && *s != 0 && *s != '=')
		*d++ = *s++;
	*d = 0;

	list = P74_download_index;
	while( list[index_a] )
	{
		if( strcasecmp(  list[index_a], name ) == 0 )   /* found ? */
			break;
		++index_a;
	}

	/* copy parameter name b */
	s = *(char**) b; d= name;
	while( *s != ' ' && *s != 0 && *s != '=')
		*d++ = *s++;
	*d = 0;

	list = P74_download_index;
	while( list[index_b] )
	{
		if( strcasecmp(  list[index_b], name ) == 0 )   /* found ? */
			break;
		++index_b;
	}

	if ( index_a <  index_b ) return -1;
	if ( index_a >  index_b ) return 1;

	return 0;
}

/* -------------------------------------------------------------------------------------
   sorts the parameter list
   -------------------------------------------------------------------------------------
*/

void sort_parameterlist( ac_inv_AxIdent *ax_ident )
{
	if( ax_ident->drive_type == 1 )
		qsort( (void*) &ax_ident->p_sorted_parameters, ax_ident->number_of_parameters, sizeof(UDINT), compare_download_index_P84 );
	else
		qsort( (void*) &ax_ident->p_sorted_parameters, ax_ident->number_of_parameters, sizeof(UDINT), compare_download_index_P74 );
}
```

#### ac_inv.c - inverter
```c
#include <bur/plctypes.h>
#include "ac_inv_global.h"

/* --------------------------------------------------------------------------------------
control the inverter
--------------------------------------------------------------------------------------
*/

//#define ETAD 			ax_ident->p_alloc->io_mapping.ETAD
#define RFRD 			ax_ident->p_alloc->io_mapping.RFRD
//#define CMDD 			ax_ident->p_alloc->io_mapping.CMDD
#define CMI				ax_ident->p_alloc->io_mapping.CMI
#define LFRD 			ax_ident->p_alloc->io_mapping.LFRD
#define MODULE_OK 		ax_ident->p_alloc->io_mapping.ModuleOK
#define _LFT			(ax_ident->p_alloc->io_mapping.LFT + ax_ident->p_alloc->io_mapping._LFT)
#define OTR				ax_ident->p_alloc->io_mapping.OTR
#define LCR				ax_ident->p_alloc->io_mapping.LCR
#define THD				ax_ident->p_alloc->io_mapping.THD
#define THR				ax_ident->p_alloc->io_mapping.THR
//#define HMIS			ax_ident->p_alloc->io_mapping.HMIS
#define LTR				ax_ident->p_alloc->io_mapping.LTR

void ac_inv(struct ac_inv* inst)
{

	UINT cmdd = 0;
	UINT etad = 0;
	UINT hmis = 0;

	if( inst->ax_ident != 0 )
	{
		ac_inv_AxIdent *ax_ident = (ac_inv_AxIdent*) inst->ax_ident;
		etad = ax_ident->p_alloc->io_mapping.ETAD;
		hmis = ax_ident->p_alloc->io_mapping.HMIS;
		ax_ident->timer += ax_ident->cycleTime;

		/* CiA 402 state machine */
		//CMDD = 0;
		LFRD = 0;
		LTR = 0;

		switch( ax_ident->step_init )
		{
		case STEP_W_NETWORK:  /* wait for network */
			inst->initialized = 0;
			if( MODULE_OK  )
			{
				inst->quickstop = 1;
				ax_ident->step_init = STEP_READ_DEVICE_NAME;
				ax_ident->fub_sdoread.pData = (UDINT) &ax_ident->device_name;
				ax_ident->fub_sdoread.datalen = sizeof(ax_ident->device_name);
				ax_ident->fub_sdoread.index = 0x1008;
				ax_ident->fub_sdoread.subindex = 0;
				ax_ident->sdo_read_step = 100; /* SDO direct read */
				ax_ident->HMIS_old = hmis +1;
			}
			break;

		case STEP_READ_DEVICE_NAME:  /* read device name */
			if( ax_ident->sdo_read_step == 0 )
			{
				if( !strcmp( ax_ident->device_name, "ACOPOS Inverter P74" ) )
					ax_ident->drive_type = 2;
				else if( !strcmp( ax_ident->device_name, "8I0IF248.300-1" ) )
					ax_ident->drive_type = 1;
				else
					ax_ident->drive_type = 0;
				ax_ident->step_init = STEP_LOG_DEVICE_TYPE;
			}
			break;

		case STEP_LOG_DEVICE_TYPE:  /* write device information into log */
		{
			char tempstring[20];

			strcpy( ax_ident->log_info, ax_ident->interface );
			strcat( ax_ident->log_info, "." );
			m_ltoa( ax_ident->node_number, tempstring, 10 );
			strcat( ax_ident->log_info, tempstring );
			strcat( ax_ident->log_info, ":" );
			strcat( ax_ident->log_info, ax_ident->device_name );
			ax_ident->fub_log_write.logLevel = arlogLEVEL_INFO;
			ax_ident->fub_log_write.errornr = 0;
			ax_ident->fub_log_write.mem = (UDINT) &ax_ident->node_number;
			ax_ident->fub_log_write.len = sizeof(ax_ident->node_number);
			ax_ident->fub_log_write.asciiString = (UDINT) ax_ident->log_info;
			AsArLogWrite( &ax_ident->fub_log_write );
			ax_ident->step_init = STEP_W_LOG_DEVICE_TYPE;
		}
		break;

		case STEP_W_LOG_DEVICE_TYPE:
			if( ax_ident->fub_log_write.status != 65535 )
			{
				if( ax_ident->drive_type == 0 )
				{
					inst->fault = 1;
					strcpy( inst->drive_state, "????" );
					strcpy( inst->fault_code, "????" );
					ax_ident->step_init = STEP_INTERNAL_ERROR;
				}
				else if( ax_ident->drive_type == 2 )    /* P74 */
				{
					CMI = 0;
					ax_ident->timer = 0;
					strcpy( ax_ident->sdo_write_par_name, "FCS" );
					strcpy( ax_ident->sdo_write_value_constant,  "InI" );
					ax_ident->sdo_write_step = 1;
					ax_ident->step_init = STEP_W_FACTORY_RESET_P74;
				}
				else    /* P84 */
				{
					ax_ident->step_init = STEP_W_FACTORY_RESET_P84;
				}
			}
			else
			{
				AsArLogWrite( &ax_ident->fub_log_write );
			}
			break;

			/* ------------------  P74 ------------------------- */

		case STEP_W_FACTORY_RESET_P74: /* wait, until factory settings done (P74) */
			if( ax_ident->sdo_write_step == 0 && ax_ident->timer > 5.0 )
			{
				CMI = 0x8000;  /* disable parameter checking */
				strcpy( ax_ident->sdo_write_par_name, "Fr1" );
				strcpy( ax_ident->sdo_write_value_constant,  "nEt" );
				ax_ident->sdo_write_step = 1;
				ax_ident->step_init = STEP_W_P74_CONFIG_1;
			}
			break;

		case STEP_W_P74_CONFIG_1:
			if( ax_ident->sdo_write_step == 0 )
			{
				strcpy( ax_ident->sdo_write_par_name, "Cd1" );
				strcpy( ax_ident->sdo_write_value_constant,  "nEt" );
				ax_ident->sdo_write_step = 1;
				ax_ident->step_init = STEP_W_P74_CONFIG_2;
			}
			break;

		case STEP_W_P74_CONFIG_2:
			if( ax_ident->sdo_write_step == 0 )
			{
				strcpy( ax_ident->sdo_write_par_name, "Cd2" );
				strcpy( ax_ident->sdo_write_value_constant,  "tEr" );
				ax_ident->sdo_write_step = 1;

				if( (etad & 0x0f) == 0x8 && _LFT == 7 )    /* "CNF" at bootup- time ? */
				{
					cmdd |= 0x80;
				}
				ax_ident->step_init = STEP_W_REFERENCE_CHANNEL_SET;
			}
			break;

			/* ------------------  P84 ------------------------- */

		case STEP_W_FACTORY_RESET_P84: /* force to factory settings (P84) */
			CMI = 1;
			ax_ident->timer = 0;
			ax_ident->step_init = STEP_W_P84_CONFIG_1;
			break;

		case STEP_W_P84_CONFIG_1:  /* wait, until factory settings done  */
			if( ax_ident->timer > 5.0 )
			{
				CMI = 0x8000;  /* disable parameter checking */
				ax_ident->timer = 0;
				ax_ident->step_init = STEP_W_P84_CONFIG_2;
			}
			break;

		case STEP_W_P84_CONFIG_2:  /* set Ref1 channel to Powerlink */
			if( ax_ident->timer > 1 )
			{
				if( ax_ident->drive_type == 2 )   /* P74 */
				{
					ax_ident->step_init = STEP_W_REFERENCE_CHANNEL_SET;
				}
				else
				{
					strcpy( ax_ident->sdo_write_par_name, "Fr1" );
					strcpy( ax_ident->sdo_write_value_constant,  "CAn" );
					ax_ident->sdo_write_step = 1;
					ax_ident->step_init = STEP_W_REFERENCE_CHANNEL_SET;
				}
			}
			break;

			/* ------------------ P74 & P84 ------------------------- */

		case STEP_W_REFERENCE_CHANNEL_SET: /* wait until reference channel is set */
			if( !MODULE_OK )
			{
				logCOF( ax_ident );
				inst->fault = 1;
				strcpy( inst->drive_state, "COF" );
				ax_ident->step_init = STEP_W_NETWORK;
				break;
			}
			if( ax_ident->sdo_write_step == 0 )
			{
				inst->status = ax_ident->sdo_write_status;
				if( inst->status == 0 )
				{
					create_parameterlist( ax_ident );
					if( ax_ident->dont_sort_parameters == 0 )
					{
						sort_parameterlist( ax_ident );
					}
					ax_ident->write_parameterlist_step = 1;
					ax_ident->step_init = STEP_W_PARAMETER_LIST_DOWNLOAD;
				}
				else
				{
					ax_ident->step_init = STEP_INTERNAL_ERROR;
				}
			}
			break;

		case STEP_W_PARAMETER_LIST_DOWNLOAD:  /* wait until parameter list is downloaded */
			if( !MODULE_OK )
			{
				logCOF( ax_ident );
				inst->fault = 1;
				strcpy( inst->drive_state, "COF" );
				ax_ident->step_init = STEP_W_NETWORK;
				break;
			}
			else   /* ready ? */
			{
				if( ax_ident->write_parameterlist_step == 0 )  /* ready ? */
				{
					inst->status = ax_ident->write_parameterlist_status;
					if( inst->status == 0 )
					{
						ax_ident->timer = 0;
						ax_ident->step_init = STEP_CHECK_PARAMETER_LIST;
					}
					else
					{
						ax_ident->step_init = STEP_INTERNAL_ERROR;
					}
				}
			}
			break;

		case STEP_CHECK_PARAMETER_LIST:
			CMI = 0; /* enable parameter checking */
			if( ax_ident->timer > 1.0 )
			{
				ax_ident->compare_parameterlist_step = 1;
				ax_ident->step_init = STEP_W_PARAMETER_LIST_CHECKED;
			}
			break;

		case STEP_W_PARAMETER_LIST_CHECKED: /* compare parameter list */
			if( !MODULE_OK )
			{
				logCOF( ax_ident );
				inst->fault = 1;
				strcpy( inst->drive_state, "COF" );
				ax_ident->step_init = STEP_W_NETWORK;
				break;
			}
			else if( ax_ident->compare_parameterlist_step == 0 ) 	/* ready ? */
			{
				inst->status = ax_ident->compare_parameterlist_status;
				if( inst->status == 0 )
				{
					ax_ident->step_init = STEP_READ_KV;
				}
				else   /* error */
				{
					ax_ident->step_init = STEP_INTERNAL_ERROR;
				}
			}
			break;

		case STEP_READ_KV: /* read kv */
			strcpy( ax_ident->sdo_read_par_name, "SPG" );
			ax_ident->sdo_read_step = 10;  /* start reading */
			ax_ident->step_init = STEP_READ_TI;
			break;

		case STEP_READ_TI: /* read ti */
			if( ax_ident->sdo_read_step == 0 )
			{
				inst->kv = ax_ident->kv_old = ax_ident->sdo_read_value;
				strcpy( ax_ident->sdo_read_par_name, "SIt" );
				ax_ident->sdo_read_step = 10;  /* start reading */
				ax_ident->step_init = STEP_READ_OUTPUT_FREQUENCY;
			}
			break;

		case STEP_READ_OUTPUT_FREQUENCY: /* read maximum output frequency  */
			if( ax_ident->sdo_read_step == 0 )
			{
				inst->ti = ax_ident->ti_old = ax_ident->sdo_read_value;
				strcpy( ax_ident->sdo_read_par_name, "tFr" );
				ax_ident->sdo_read_step = 10;  /* start reading */
				ax_ident->step_init = STEP_READ_TORQUE_LIMIT_0;
			}
			break;

		case STEP_READ_TORQUE_LIMIT_0: /* read motor torque limitation 0  */
			if( ax_ident->sdo_read_step == 0 )
			{
				ax_ident->maximum_output_frequency = (REAL) ax_ident->sdo_read_value / 10.0;
				strcpy( ax_ident->sdo_read_par_name, "tLIM" );
				ax_ident->sdo_read_step = 10;  /* start reading */
				ax_ident->step_init = STEP_READ_TORQUE_LIMIT_1;
			}
			break;

		case STEP_READ_TORQUE_LIMIT_1: /* read motor torque limitation 1  */
			if( ax_ident->sdo_read_step == 0 )
			{
				inst->t_limit[0] = ax_ident->t_limit_old[0] = (REAL) ax_ident->sdo_read_value;
				strcpy( ax_ident->sdo_read_par_name, "tLIG" );
				ax_ident->sdo_read_step = 10;  /* start reading */
				ax_ident->step_init = STEP_READ_CTT;
			}
			break;

		case STEP_READ_CTT: /* read Ctt  */
			if( ax_ident->sdo_read_step == 0 )
			{
				inst->t_limit[1] = ax_ident->t_limit_old[1] = (REAL) ax_ident->sdo_read_value;
				strcpy( ax_ident->sdo_read_par_name, "Ctt" );
				ax_ident->sdo_read_step = 10;  /* start reading */
				ax_ident->step_init = STEP_READ_RATED_FREQ;
			}
			break;

		case STEP_READ_RATED_FREQ: /* read rated motor frequency  or torque  */
			if( ax_ident->sdo_read_step == 0 )
			{
				if( ax_ident->sdo_read_value == 5 )   /* 5 = "SyN" */
				{
					ax_ident->use_rpm = 1;
					ax_ident->step_init = STEP_W_COMMAND;
				}
				else   /* only allowed for induction motors */
				{
					strcpy( ax_ident->sdo_read_par_name, "FrS" );
					ax_ident->sdo_read_step = 10;  /* start reading */
					ax_ident->step_init = STEP_READ_RATED_SPEED;
				}
			}
			break;

		case STEP_READ_RATED_SPEED: /* read rated motor speed  */
			if( ax_ident->sdo_read_step == 0 )
			{
				ax_ident->rated_motor_frequency = (REAL) ax_ident->sdo_read_value / 10.0;
				strcpy( ax_ident->sdo_read_par_name, "nSP" );
				ax_ident->sdo_read_step = 10;  /* start reading */
				ax_ident->step_init = STEP_W_READ_RATED_SPEED;
			}
			break;

		case STEP_W_READ_RATED_SPEED: /* wait until read  */
			if( ax_ident->sdo_read_step == 0 )
			{
				ax_ident->rated_motor_speed = (REAL) ax_ident->sdo_read_value;
				ax_ident->polepairs = 60.0 * ax_ident->rated_motor_frequency	/ ax_ident->rated_motor_speed;
				ax_ident->HMIS_old = 0xffff;
				ax_ident->step_init = STEP_W_COMMAND;
			}
			break;

		/* ---------------------------------------------------
			drive is initialized
			-------------------------------------------------- */

		case STEP_W_COMMAND:  /* initialization successful */
			inst->initialized = 1;
			if( !MODULE_OK )
			{
				logCOF( ax_ident );
				inst->fault = 1;
				strcpy( inst->drive_state, "COF" );
				inst->initialized = 0;
				ax_ident->step_init = STEP_W_NETWORK;
			}
			else
			{
				if( inst->quickstop && inst->activate_tuning && inst->ctrl_is_on == 0 && inst->ctrl_on == 1 && ax_ident->drive_type == 1 )
				{
					ax_ident->ctrl_on_internal = 0;
					strcpy( ax_ident->sdo_write_par_name, "tUn" );
					strcpy( ax_ident->sdo_write_value_constant,  "yES" );
					ax_ident->sdo_write_step = 1;
					ax_ident->step_init = STEP_P84_WRITE_TUN;
				}
				else if( inst->quickstop && inst->activate_tuning && inst->ctrl_is_on == 0 && inst->ctrl_on == 1 && ax_ident->drive_type == 2 )
				{
					ax_ident->ctrl_on_internal = 0;
					ax_ident->timer = 0;
					ax_ident->step_init = STEP_P74_START_TUNING;
				}
				else
				{
					ax_ident->ctrl_on_internal = inst->ctrl_on;
				}

			}
			break;

		case STEP_P84_WRITE_TUN:
			if( !MODULE_OK )
			{
				logCOF( ax_ident );
				inst->fault = 1;
				strcpy( inst->drive_state, "COF" );
				ax_ident->step_init = STEP_W_NETWORK;
			}
			else if( ax_ident->sdo_write_step == 0 )
			{
				ax_ident->ctrl_on_internal = 1;
				ax_ident->step_init = STEP_W_P84_TUNING_DONE;
			}
			break;

		case STEP_W_P84_TUNING_DONE:
			if( !MODULE_OK )
			{
				logCOF( ax_ident );
				inst->fault = 1;
				strcpy( inst->drive_state, "COF" );
				ax_ident->step_init = STEP_W_NETWORK;
			}
			else if( inst->ctrl_is_on )
			{
				ax_ident->step_init = STEP_W_COMMAND;
			}
			break;

		case STEP_P74_START_TUNING:
		    ax_ident->tempUINT = (1<<8);  /* Halt */
			cmdd = ax_ident->tempUINT;
			ax_ident->timer = 0;
			ax_ident->step_init = STEP_P74_TUNING_1;
			break;

		case STEP_P74_TUNING_1:
			if( ax_ident->timer > 0.1 )
			{
			    ax_ident->tempUINT |= (1<<1);  /* enable voltage */
				ax_ident->timer = 0;
				ax_ident->step_init = STEP_P74_TUNING_2;
			}
			cmdd = ax_ident->tempUINT;
			break;

		case STEP_P74_TUNING_2:
			if( etad & (1<<4) )  /* voltage enabled ? */
			{
			    ax_ident->tempUINT |= (1<<2);   /* no quickstop */
				ax_ident->timer = 0;
				ax_ident->step_init = STEP_P74_TUNING_3;
			}
			cmdd = ax_ident->tempUINT;
			break;

		case STEP_P74_TUNING_3:
			if( ax_ident->timer > 0.1 )
			{
			    ax_ident->tempUINT |= (1<<0);   /* switch on */
				ax_ident->timer = 0;
				ax_ident->step_init = STEP_P74_TUNING_4;
			}
			cmdd = ax_ident->tempUINT;
			break;

		case STEP_P74_TUNING_4:
			if( (etad & (1<<0)) || (ax_ident->timer > 1.0) )  /* read to switch on ? */
			{
			    ax_ident->tempUINT |= (1<<3);   /* enable operation */
				ax_ident->timer = 0;
				ax_ident->step_init = STEP_P74_TUNING_5;
			}
			cmdd = ax_ident->tempUINT;
			break;

		case STEP_P74_TUNING_5:
			if( (etad & (2<<0)) || (ax_ident->timer > 1.0) )  /* switched on ? */
			{
				strcpy( ax_ident->sdo_write_par_name, "tUn" );
				strcpy( ax_ident->sdo_write_value_constant,  "yES" );
				ax_ident->sdo_write_step = 1;
				ax_ident->timer = 0;
				ax_ident->step_init = STEP_P74_TUNING_6;
			}
			cmdd = ax_ident->tempUINT;
			break;

		case STEP_P74_TUNING_6:
			if( ax_ident->sdo_write_step == 0 || (ax_ident->timer > 1.0) )  /* parameter downloaded ? */
			{
				ax_ident->tempUINT &= ~(1<<8); /* no halt */
				ax_ident->ctrl_on_internal = 1;
				ax_ident->timer = 0;
				ax_ident->step_init = STEP_P74_TUNING_7;
			}
			cmdd = ax_ident->tempUINT;
			break;

		case STEP_P74_TUNING_7:
			if( (ax_ident->timer > 0.5) && (hmis != 0) ) /* tuning done ? */
			{
				ax_ident->step_init = STEP_P74_TUNING_8;
			}
			cmdd = ax_ident->tempUINT;
			break;

		case STEP_P74_TUNING_8:
			if( !MODULE_OK )
			{
				logCOF( ax_ident );
				inst->fault = 1;
				strcpy( inst->drive_state, "COF" );
				ax_ident->step_init = STEP_W_NETWORK;
			}
			else if( inst->ctrl_is_on )
			{
				ax_ident->step_init = STEP_W_COMMAND;
			}
			break;

		case STEP_INTERNAL_ERROR: /* error */
			if( !MODULE_OK )
			{
				logCOF( ax_ident );
				inst->fault = 1;
				strcpy( inst->drive_state, "COF" );
				ax_ident->step_init = 0;
				break;
			}
			inst->fault = 1;
			break;

		}

		/* Power removal */
		if( ax_ident->ctrl_on_internal == 0 )
		{
			inst->PRA_detected = 0;
		}
		if( hmis == 12 )  /* PrA - Power removal */
		{
			inst->PRA_detected = 1;
		}

		/* CiA 402 state machine */

		inst->ctrl_is_on = 0;
		if( inst->initialized )
		{
			if( ax_ident->ctrl_on_internal && !inst->PRA_detected )
			{
				if( (etad & 0xfe) == 0x40 || (etad & 0xfe) == 0x50 )   /* switch on disabled */
				{
					cmdd = 0x6;
					/*LFRD = 0;*/
					inst->ctrl_is_on = 0;
					/*strcpy( inst->drive_state, "nSt" );*/
				}
				else if( (etad & 0xff) == 0x21 || (etad & 0xff) == 0x31 )   /* ready to switch on */
				{
					cmdd = 0x7;
					/*LFRD = 0;*/
					inst->ctrl_is_on = 0;
					/*
					if( (ETAD & 0xff) == 0x21 )
					strcpy( inst->drive_state, "nSt" );
					else if( (ETAD & 0xff) == 0x31 )
					strcpy( inst->drive_state, "rDY" );
					*/
				}
				else if( (etad & 0xff) == 0x33   )   /* switched on */
				{
					cmdd = 0xf;
					/*LFRD = 0;*/
					inst->ctrl_is_on = 1;
					/*strcpy( inst->drive_state, "rDY" );				*/
				}
				else if( (etad & 0xff) == 0x37  )   /* movement enabled */
				{
					cmdd = 0xf;
					if( ax_ident->use_rpm )
					{
						LFRD = (INT) inst->n_set;
					}
					else
					{
						LFRD = (INT)((inst->n_set * 60.0 * ax_ident->maximum_output_frequency)/(100.0 *ax_ident->polepairs));
					}
					LTR = (INT) (inst->t_set * 10.0);
					inst->ctrl_is_on = 1;
					/*strcpy( inst->drive_state, "rUn" );								*/
				}

			}

		} /* end of if( inst->initialized ) ... */
		if( !inst->quickstop )
			cmdd = 0x0002;
		if( inst->C211 )
			cmdd |= 0x0800;
		if( inst->C212 )
			cmdd |= 0x1000;
		if( inst->C213 )
			cmdd |= 0x2000;
		if( inst->C214 )
			cmdd |= 0x4000;
		if( inst->C215 )
			cmdd |= 0x8000;

		if( inst->initialized || inst->fault )
		{

			/* actual values */
			if( ax_ident->use_rpm )
			{
				inst->n_act = RFRD;
			}
			else
			{
				if( ax_ident->maximum_output_frequency > 0.0001 )
					inst->n_act = (100.0 * (REAL) RFRD * ax_ident->polepairs) / (ax_ident->maximum_output_frequency * 60.0);
				else
					inst->n_act = 0.0;
			}
			inst->alarm = etad & 0x80 ? 1 : 0;
			inst->fault = (etad & 0x0f) == 0x8 ? 1 : 0;
			inst->LFT = _LFT;
			inst->current = (REAL) LCR * 0.1;
			inst->t_act = (REAL) OTR * 0.1;
			inst->thst_drive = (REAL) THD;
			inst->thst_motor = (REAL) THR;

			/* drive state */
			if( hmis != ax_ident->HMIS_old )
			{
				char *s;
				ax_ident->HMIS_old = hmis;
				s = find_value_constant( "HMIS", hmis, ax_ident->drive_type );
				if( s )
					strncpy( inst->drive_state, s, 4 );
			}

			/* fault code */
			if( inst->fault )
			{
				char *s;
				s = find_value_constant( "LFT", _LFT, ax_ident->drive_type );
				if( s )
				{
					strncpy( inst->fault_code, s, 4 );
				}
			}
			else
			{
				memset( inst->fault_code, 0, sizeof(inst->fault_code) );
			}

			/* quit faults */
			if( inst->f_quit )
			{
				cmdd |= 0x80;
			}

			switch( ax_ident->step_read_data )
			{
			case 0: /* wait for command */
				++ax_ident->counter_cyclic_data;
				if( inst->read_parameter == 1 )
				{
					inst->read_parameter = 2; /* busy */
					strcpy( ax_ident->sdo_read_par_name, inst->parameter_name );
					ax_ident->sdo_read_step = 1;  /* start reading */
					ax_ident->step_read_data = 10; /* let user read data from drive */
				}
				else if( ax_ident->counter_cyclic_data > 10 )   /* read cylic fub data */
				{
					strcpy( ax_ident->sdo_read_par_name, "ULN" );
					ax_ident->sdo_read_step = 10;  /* start reading (without logging) */
					ax_ident->step_read_data = 20;
				}
				break;

			case 10: /* let user read data from drive */
				if( ax_ident->sdo_read_step == 0 )
				{
					if( ax_ident->sdo_read_status )
					{
						char tempstring[20];
						inst->status = ax_ident->sdo_read_status;
						m_ltoa( ax_ident->sdo_read_errorinfo, tempstring, 16 );
						strcpy( inst->parameter_value, "16#" );
						strcat( inst->parameter_value, tempstring );
					}
					else
					{
						inst->status = 0;
						strcpy( inst->parameter_value, ax_ident->sdo_read_value_constant );
					}
					inst->read_parameter = 0;
					ax_ident->step_read_data = 0;
				}
				break;

			case 20: /* read cyclic data from drive */
				if( ax_ident->sdo_read_step == 0 )
				{
					if( ax_ident->sdo_read_status == 0)
					{
						inst->udc = (REAL)ax_ident->sdo_read_value / 10.0 * 1.414213;
					}
					if( ax_ident->drive_type == 1 )   /* P84 */
					{
						strcpy( ax_ident->sdo_read_par_name, "PUC" );
						ax_ident->sdo_read_step = 10;  /* start reading (without logging) */
						ax_ident->step_read_data = 21;
					}
					else    /* P74 */
					{
						ax_ident->step_read_data = 0;
						ax_ident->counter_cyclic_data = 0;
					}
				}
				break;

			case 21: /* */
				if( ax_ident->sdo_read_step == 0 )
				{
					if( ax_ident->sdo_read_status == 0)
					{
						inst->encoder_value = (UINT) ax_ident->sdo_read_value;
					}
					ax_ident->step_read_data = 0;
					ax_ident->counter_cyclic_data = 0;
				}
				break;

			} /* end of switch( ax_ident->step_read_data )... */

			/* write a parameter to inverter */
			if( inst->write_parameter == 1 && ax_ident->sdo_write_step == 0 )
			{
				inst->write_parameter = 2;
			}
			if( inst->write_parameter == 2 && ax_ident->sdo_write_step == 0 )
			{
				strcpy( ax_ident->sdo_write_par_name, inst->parameter_name );
				strcpy( ax_ident->sdo_write_value_constant, inst->parameter_value );
				inst->write_parameter = 3;
				ax_ident->sdo_write_step = 1; /* start writing */
			}
			if( inst->write_parameter == 3 && ax_ident->sdo_write_step == 0 )
			{
				inst->status = 0;
				if( ax_ident->sdo_write_status )
				{
					char tempstring[20];
					inst->status = ax_ident->sdo_write_status;
					m_ltoa( ax_ident->sdo_write_errorinfo, tempstring, 16 );
					strcpy( inst->parameter_value, "16#" );
					strcat( inst->parameter_value, tempstring );
				}
				inst->write_parameter = 0;
			}

			/* write new kv to inverter */
			if( (inst->write_parameter == 0) && (inst->kv != ax_ident->kv_old ) && ax_ident->sdo_write_step == 0 )
			{
				ax_ident->kv_old = inst->kv;
				strcpy( inst->parameter_name, "SPG" );
				m_ltoa( inst->kv, (char*) inst->parameter_value, 10 );
				inst->write_parameter = 1;
			}

			/* write new ti to inverter */
			if( (inst->write_parameter == 0) && (inst->ti != ax_ident->ti_old ) && ax_ident->sdo_write_step == 0 )
			{
				ax_ident->ti_old = inst->ti;
				strcpy( inst->parameter_name, "SIt" );
				m_ltoa( inst->ti, (char*) inst->parameter_value, 10 );
				inst->write_parameter = 1;
			}

			/* write new motoring torque limitation to inverter */
			if( (inst->write_parameter == 0) && (fabs( inst->t_limit[0] - ax_ident->t_limit_old[0]) >= 0.1 ) && ax_ident->sdo_write_step == 0 )
			{
				ax_ident->t_limit_old[0] = inst->t_limit[0];
				strcpy( inst->parameter_name, "tLIM" );
				m_ltoa( inst->t_limit[0], (char*) inst->parameter_value, 10 );
				inst->write_parameter = 1;
			}

			/* write new generatoring torque limitation to inverter */
			if( (inst->write_parameter == 0) && (fabs( inst->t_limit[1] - ax_ident->t_limit_old[1]) >= 0.1 ) && ax_ident->sdo_write_step == 0 )
			{
				ax_ident->t_limit_old[1] = inst->t_limit[1];
				strcpy( inst->parameter_name, "tLIG" );
				m_ltoa( inst->t_limit[1], (char*) inst->parameter_value, 10 );
				inst->write_parameter = 1;
			}

		}  /* end of if( inst->initialized || inst->fault )... */

		/* call subroutines */
		if( MODULE_OK )
		{
			write_parameterlist( ax_ident );
			compare_parameterlist( ax_ident );
			read_parameter( ax_ident );
			write_parameter( ax_ident );
		}

		inst->power_line = etad & 0x10 ? 1 : 0;
		inst->ctrl_ready = inst->initialized && inst->power_line && !inst->fault && inst->quickstop;

 		ax_ident->p_alloc->io_mapping.CMDD = cmdd;

	}
	else
	{
		inst->status = ac_invlibERR_ILLEGAL_AXIDENT;
	}

}

void logCOF( ac_inv_AxIdent *ax_ident )
{
	char tempstring1[80];
	char tempstring2[20];
	strcpy( tempstring1, "ac_invlib COF node " );
	m_ltoa( ax_ident->node_number, tempstring2, 10 );
	strcat( tempstring1, tempstring2 );
	ERRxwarning( ac_invlibERR_NETWORK, ax_ident->step_init, tempstring1 );
}
```

#### ac_inv_alloc.c
```c
/********************************************************************
 * COPYRIGHT -- Bernecker + Rainer
 ********************************************************************
 * Library: ac_invlib
 * File: ac_inv_alloc.c
 * Author: hilchenbachc
 * Created: December 16, 2009
 *******************************************************************/

#include <bur/plctypes.h>
#include "ac_inv_global.h"

/* -----------------------------------------------------------------------------------
axis allocation
-----------------------------------------------------------------------------------
*/

void ac_inv_alloc( struct ac_inv_alloc* inst ){
	ac_inv_AxIdent *ax_ident;
	char *token;
	struct EplGetLocalNodeID fub_getlocalnodeid;
	struct CANopenGetLocalNodeID fub_canopen_getlocalnodeid;
	RTInfo_typ rt_info;

	/* check version of Automation Runtime */
	{
		struct TARGETInfo fub_targetinfo;
		char   v[7];
		long   version;

		fub_targetinfo.enable = 1;
		fub_targetinfo.pOSVersion = (UDINT) &v;
		TARGETInfo( &fub_targetinfo );
		version = v[0]-'A' + 1000 * (v[2]-'0') + 100 * (v[4]-'0') + 10 * (v[5]-'0');
		if( version < 2963 ){
			ERRxfatal( ac_invlibERR_WRONG_ARVERSION, 0, "ACPinverter: AR >= D2.96 required" );
			return;
		}
	}

	inst->status = TMP_alloc( sizeof(ac_inv_AxIdent), (void*) &inst->ax_ident );
	if( inst->status == 0 ){
		memset( (void*) inst->ax_ident, 0, sizeof(ac_inv_AxIdent) );

		ax_ident = (ac_inv_AxIdent *) inst->ax_ident;
		ax_ident->p_alloc = inst;

		if( inst->pDevice ){
			char device[40];
			strcpy( device, (char*) inst->pDevice );

			token = strtok( device , "." );
			while( token != NULL )
			{
				if( !strncmp( token, "ST", 2 ) ){
					if( strlen(token) >=3 ){
						ax_ident->node_number = m_atol( token+2 );
					}
					else {
						inst->status = ERR_ASEPL_WRONG_DEVICE;
						inst->ax_ident = 0;
						return;
					}
				}
				else if( !strncmp( token, "IF", 2 ) ){
					if( strlen(token) >= 3 ){
						char *p = strstr( (char*) inst->pDevice, "IF" );
						strncpy( ax_ident->interface, (char*) inst->pDevice, (UDINT) p - inst->pDevice );
						strcat( ax_ident->interface, token );
					}
					else {
						inst->status = ERR_ASEPL_WRONG_DEVICE;
						inst->ax_ident = 0;
						return;
					}
				}
				token = strtok(NULL, "." );
			}

		}
		else {
			strcpy( inst->message, "Wrong device name !" );
			inst->status = ERR_ASEPL_WRONG_DEVICE;
			inst->ax_ident = 0;
			return;
		}

	}
	else {
		strcpy( inst->message, "Error at TMP_alloc()" );
		inst->ax_ident = 0;
		return;
	}

	/* check device name */
	memset( &fub_getlocalnodeid, 0, sizeof(fub_getlocalnodeid) );
	fub_getlocalnodeid.enable = 1;
	fub_getlocalnodeid.pDevice = (plcstring*) ax_ident->interface;

	memset( &fub_canopen_getlocalnodeid, 0, sizeof(fub_canopen_getlocalnodeid) );
	fub_canopen_getlocalnodeid.enable = 1;
	fub_canopen_getlocalnodeid.pDevice = (UDINT) ax_ident->interface;

	ax_ident->isCANopen = 0;

	do {
		EplGetLocalNodeID( &fub_getlocalnodeid );
	} while( fub_getlocalnodeid.status == 65535 );
	inst->status = 	fub_getlocalnodeid.status;

	if( inst->status == ERR_ASEPL_WRONG_DEVICE ){

		do {
			CANopenGetLocalNodeID( &fub_canopen_getlocalnodeid );
		} while( fub_canopen_getlocalnodeid.status == 65535 );
		inst->status = 	fub_canopen_getlocalnodeid.status;

		if( inst->status == ERR_CANOPEN_DEVICE_NOT_FOUND || inst->status == ERR_CANOPEN_DEVICE_NOT_OPENED ){
			strcpy( inst->message, "device is not a valid EPL oder CANopen node" );
			inst->ax_ident = 0;
			return;
		}
		else if( inst->status != 0 ){
			strcpy( inst->message, "Error at CANopenGetLocalNodeID()" );
			inst->ax_ident = 0;
			return;
		}
		ax_ident->isCANopen = 1;

	}
	else if( inst->status != 0 ){
		strcpy( inst->message, "Error at EplGetLocalNodeID()" );
		inst->ax_ident = 0;
		return;
	}

	ax_ident->use_rpm = inst->rpm;
	ax_ident->dont_sort_parameters = inst->no_parameter_sort;

  	rt_info.enable = 1;     /* enables the function */
	RTInfo(&rt_info);       /* gets information from the software object */
	ax_ident->cycleTime = (REAL) rt_info.cycle_time / 1.0e6;

	/* initialize SDO fubs */
	if( ax_ident->isCANopen ){
		memset( &ax_ident->fub_canopen_sdoread, 0, sizeof(ax_ident->fub_canopen_sdoread) );
		ax_ident->fub_canopen_sdoread.pDevice = (UDINT) ax_ident->interface;
		ax_ident->fub_canopen_sdoread.node = ax_ident->node_number;
	    ax_ident->fub_canopen_sdoread.pRxdata = (UDINT) &ax_ident->sdo_read_value;
		ax_ident->fub_canopen_sdoread.maxlength = sizeof(ax_ident->sdo_read_value);

		memset( &ax_ident->fub_canopen_sdowrite, 0, sizeof(ax_ident->fub_canopen_sdowrite) );
		ax_ident->fub_canopen_sdowrite.pDevice = (UDINT) ax_ident->interface;
		ax_ident->fub_canopen_sdowrite.node = ax_ident->node_number;
		ax_ident->fub_canopen_sdowrite.pTxdata = (UDINT) &ax_ident->sdo_write_value;
		ax_ident->fub_canopen_sdowrite.txlength = sizeof(ax_ident->sdo_write_value);
	}
	else {
		memset( &ax_ident->fub_sdoread, 0, sizeof(ax_ident->fub_sdoread) );
		ax_ident->fub_sdoread.pDevice = (plcstring*) ax_ident->interface;
		ax_ident->fub_sdoread.node = ax_ident->node_number;
	    ax_ident->fub_sdoread.pData = (UDINT) &ax_ident->sdo_read_value;
		ax_ident->fub_sdoread.datalen = sizeof(ax_ident->sdo_read_value);

		memset( &ax_ident->fub_sdowrite, 0, sizeof(ax_ident->fub_sdowrite) );
		ax_ident->fub_sdowrite.pDevice = (plcstring*) ax_ident->interface;
		ax_ident->fub_sdowrite.node = ax_ident->node_number;
		ax_ident->fub_sdowrite.pData = (UDINT) &ax_ident->sdo_write_value;
		ax_ident->fub_sdowrite.datalen = sizeof(ax_ident->sdo_write_value);
	}

	/* check if data objects available */
	{
		int i;

		for( i = 0; i < (sizeof(inst->pcfgpar)/sizeof(inst->pcfgpar[0])); ++i ){
			memset( &ax_ident->fub_datobjinfo, 0, sizeof(ax_ident->fub_datobjinfo) );
			ax_ident->fub_datobjinfo.enable = 1;
			if( inst->pcfgpar[i]){
				ax_ident->fub_datobjinfo.pName = inst->pcfgpar[i];
				DatObjInfo( &ax_ident->fub_datobjinfo	);
				inst->status = ax_ident->fub_datobjinfo.status;
				if( inst->status == doERR_MODULNOTFOUND ){
					strcpy( inst->message, "module not found: \"" );
					strcat( inst->message, (char*) ax_ident->fub_datobjinfo.pName );
					strcat( inst->message, "\"" );
					inst->ax_ident = 0;
					return;
				}
				else if( inst->status ){
					strcpy( inst->message, "Error at DatObjInfo(\"" );
					strcat( inst->message, (char*) ax_ident->fub_datobjinfo.pName );
					strcat( inst->message, "\")" );
					inst->ax_ident = 0;
					return;
				}
			}
		}
	}

	/* access log */
	{
		struct AsArLogCreate fub_logcreate;
		struct AsArLogGetInfo fub_loginfo;

		memset( &fub_loginfo, 0, sizeof(fub_loginfo) );
		fub_loginfo.enable = 1;
		fub_loginfo.pName = (UDINT) "ac_invlog";
		do {
			AsArLogGetInfo( &fub_loginfo );
		} while( fub_loginfo.status == 65535 );
		if( fub_loginfo.status == 0 ){
			ax_ident->fub_log_write.ident = fub_loginfo.ident;
		}
		else if( fub_loginfo.status == arlogERR_NOTEXISTING ){  /* module doesn't exist */
			/* create log */
			memset( &fub_logcreate, 0, sizeof(fub_logcreate) );
			fub_logcreate.enable = 1;
			fub_logcreate.pName = fub_loginfo.pName;
			fub_logcreate.len = 128*1024;
			fub_logcreate.memType = arlogDRAM;
			do {
				AsArLogCreate( &fub_logcreate );
			} while( fub_logcreate.status == 65535 );
			if( fub_logcreate.status == 0 ){
				ax_ident->fub_log_write.ident = fub_logcreate.ident;
			}
			else {
				inst->status = fub_logcreate.status;
				strcpy( inst->message, "Error at AsArLogCreate()" );
				inst->ax_ident = 0;
				return;
			}
		}
		else { /* other errors */
			inst->status = fub_loginfo.status;
			strcpy( inst->message, "Error at AsArLogGetInfo()" );
			inst->ax_ident = 0;
			return;
		}
		ax_ident->fub_log_write.enable = 1;
	}

}
```

#### ac_invparameter.h
```c
/********************************************************************
 * COPYRIGHT -- Bernecker + Rainer
 ********************************************************************
 * Bibliothek: ac_invlib
 * Datei: ac_invparameter.h
 * Autor: hilchenbachc
 * Erstellt: 11. April 2014
 *******************************************************************/

#include <bur/plctypes.h>

typedef struct {
	char 		*name;
	INT			value;
} acpienumeration;

typedef struct {
	char 		*name;    		/* name of register */
	UINT		index;			/* CANopen index */
	USINT		subindex;		/* CANopen subindex */
	USINT		sign;
	acpienumeration *enu;		/* Value - Enumeration */
} acpireg;
```
